// This function has been automatically generated from the project information.
VAR_GLOBAL CONSTANT
	{attribute 'const_non_replaced'}
	stLibVersion_Sqlite_Adaptor : ST_LibVersion := (iMajor := 1, iMinor := 0, iBuild := 0, iRevision := 0, sVersion := '1.0');
END_VAR

(* stored: Version 1.1.0.1, ProductVersion 3.1.0.36
   GVL Global_Version: Id {a76abb3a-f19d-4cf1-a167-b69f12a8dbb3} *)
